(* IEC 61131-3 sources: Word/plc-course/02-electrical-and-field-devices/labs/solutions, 3 files *)

(* ---- 02-1-fail-safe-motor.st ---- *)
(* Lab 02-1: Fail-safe motor circuit - NC stop and overload contacts.
   Module 02 (Electrical fundamentals and field devices).
   REFERENCE SOLUTION - try the lab yourself first.
   Training exercise only: a real machine's emergency stop and safety
   functions are hard-wired or use safety-rated devices (Module 20). *)

PROGRAM FailSafeMotor
  VAR (* I/O - addresses follow the OpenPLC convention *)
    StartPB       AT %IX0.0 : BOOL;  (* Start push-button -S2, NO: TRUE while pressed *)
    StopPB_NC     AT %IX0.1 : BOOL;  (* Stop push-button -S1, NC: TRUE while NOT pressed *)
    OverloadOK_NC AT %IX0.2 : BOOL;  (* Overload relay -F2 contact 95-96, NC: TRUE while healthy *)
    Motor         AT %QX0.0 : BOOL;  (* Motor contactor -Q1 coil (through an interposing relay) *)
    TripLamp      AT %QX0.1 : BOOL;  (* Amber "overload tripped" lamp -H2 *)
  END_VAR

  (* Both NC inputs read TRUE when everything is healthy. A pressed button, a
     tripped overload, a broken wire, a loose terminal or a blown fuse all make
     them read FALSE, so every one of those faults stops the motor. That is
     the point of NC wiring: the "healthy" state has to be actively proven by
     current flowing, so any break in the circuit fails safe.

     Seal-in with both stop conditions in series (AND) with the whole rung:
     when either NC input goes FALSE, Motor drops out and the seal-in is lost.
     When the overload is reset later, nothing restarts: Motor is FALSE and
     only a fresh press of Start can set it again. *)
  Motor := (StartPB OR Motor) AND StopPB_NC AND OverloadOK_NC;

  (* The lamp shows the overload (or its wiring) is not healthy. *)
  TripLamp := NOT OverloadOK_NC;
END_PROGRAM

CONFIGURATION Config0
  RESOURCE Res0 ON PLC
    TASK MainTask(INTERVAL := T#10ms, PRIORITY := 0);
    PROGRAM Inst0 WITH MainTask : FailSafeMotor;
  END_RESOURCE
END_CONFIGURATION

(* ---- 02-2-solenoid-valves.st ---- *)
(* Lab 02-2: Solenoid valves - single-solenoid spring-return versus
   double-solenoid (bistable) valves on the same transfer line.
   Module 02 (Electrical fundamentals and field devices).
   REFERENCE SOLUTION - try the lab yourself first.
   Training exercise only: a real high-high level trip is a safety function
   and would be engineered separately (Module 20). *)

PROGRAM SolenoidValves
  VAR (* I/O - addresses follow the OpenPLC convention *)
    OpenPB         AT %IX0.0 : BOOL;  (* "Open line" push-button, NO: TRUE while pressed *)
    ClosePB_NC     AT %IX0.1 : BOOL;  (* "Close line" push-button, NC: TRUE while NOT pressed *)
    HighLevelOK_NC AT %IX0.2 : BOOL;  (* LSHH on the receiving tank, NC: TRUE while level is NOT high-high *)
    XV201_Sol      AT %QX0.0 : BOOL;  (* XV-201 solenoid: single-solenoid, spring return, fail closed *)
    XV202_OpenSol  AT %QX0.1 : BOOL;  (* XV-202 "open" coil: double-solenoid valve, stays put (fail last) *)
    XV202_CloseSol AT %QX0.2 : BOOL;  (* XV-202 "close" coil *)
  END_VAR
  VAR (* internal *)
    LineOpenCmd : BOOL;  (* TRUE = the line should be open *)
  END_VAR

  (* One command for the line, with a seal-in. Close and the high-high trip
     are NC inputs in series, so a pressed button, a high-high level or a
     broken wire all drop the command. When the trip clears, the command stays
     FALSE until an operator presses Open again: no automatic re-opening. *)
  LineOpenCmd := (OpenPB OR LineOpenCmd) AND ClosePB_NC AND HighLevelOK_NC;

  (* Single-solenoid, spring-return valve: energised = open. The output must
     stay on for as long as the valve is to be open; removing it (by the
     program, by the PLC stopping, or by a power cut) lets the spring close
     the valve. That is why this valve type is used for trips. *)
  XV201_Sol := LineOpenCmd;

  (* Double-solenoid valve: de-energising a coil does NOT move it. The PLC must
     actively drive the close coil to close it. Maintained signals are used:
     the coil for the commanded position stays energised, which re-asserts the
     position if someone has used the manual override, and the two coils are
     complementary, so they can never both be on. At power-up LineOpenCmd is
     FALSE, so the PLC drives the valve closed: after a power cut the program
     cannot know where the valve was left. *)
  XV202_OpenSol  := LineOpenCmd;
  XV202_CloseSol := NOT LineOpenCmd;
END_PROGRAM

CONFIGURATION Config0
  RESOURCE Res0 ON PLC
    TASK MainTask(INTERVAL := T#10ms, PRIORITY := 0);
    PROGRAM Inst0 WITH MainTask : SolenoidValves;
  END_RESOURCE
END_CONFIGURATION

(* ---- 02-3-namur-line-fault.st ---- *)
(* Lab 02-3: NAMUR sensor with line-fault detection - turn a switching
   signal plus open-circuit and short-circuit status bits into a validated
   signal and a fault.
   Module 02 (Electrical fundamentals and field devices).
   REFERENCE SOLUTION - try the lab yourself first.
   Training exercise only: this LSH is a control function. An independent
   high-high protection layer would be engineered separately (Module 20). *)

PROGRAM NamurLineFault
  VAR (* I/O - addresses follow the OpenPLC convention *)
    FillSel      AT %IX0.0 : BOOL;  (* Fill selector: TRUE = operator wants the tank filled *)
    SensorOn     AT %IX0.1 : BOOL;  (* LSH-301 via isolator: TRUE = NAMUR current in the ON band = fork dry *)
    WireBreak    AT %IX0.2 : BOOL;  (* Isolator status: open circuit detected (TRUE = fault) *)
    ShortCircuit AT %IX0.3 : BOOL;  (* Isolator status: short circuit detected (TRUE = fault) *)
    ResetPB      AT %IX0.4 : BOOL;  (* Fault reset push-button, NO: TRUE while pressed *)
    InletValve   AT %QX0.0 : BOOL;  (* XV-301 inlet valve solenoid, spring return: TRUE = open *)
    FaultLamp    AT %QX0.1 : BOOL;  (* Amber "LSH-301 line fault" lamp, latched *)
  END_VAR
  VAR (* internal - required by the lab interface *)
    LineFault : BOOL;  (* TRUE while an open or short circuit is present *)
    HighLevel : BOOL;  (* validated high level: TRUE when high OR when the signal cannot be trusted *)
  END_VAR

  (* 1. Signal quality. Either line fault means SensorOn cannot be trusted:
        a broken wire gives no current (reads as "wet"), and a short circuit
        gives a high current (reads as "dry", the DANGEROUS direction). *)
  LineFault := WireBreak OR ShortCircuit;

  (* 2. Validated signal. The fork is set up fail-safe: current flows while it
        is dry, so a dead sensor reads "wet" = high level. On a line fault the
        program substitutes the safe value, high level, instead of using
        SensorOn. *)
  HighLevel := (NOT SensorOn) OR LineFault;

  (* 3. Latched fault lamp. The fault sets the lamp (and wins while it is
        present). Reset clears it only after the fault has gone, so a brief
        or intermittent fault is still visible to the operator later. *)
  FaultLamp := LineFault OR (FaultLamp AND NOT ResetPB);

  (* 4. Control: fill only when asked to, when the level is known to be below
        the switch, and when no line fault is waiting to be reset.
        - A real high level is a process condition: when the level falls below
          the fork again, filling resumes by itself (a permissive).
        - A line fault is an equipment problem: filling stays stopped until
          someone has looked at it and pressed Reset. That also stops a loose
          terminal from making the valve chatter.
        FaultLamp is worked out above, before it is used here, so the valve
        responds to a reset in the same scan (Module 01: order the program in
        the direction the data flows). *)
  InletValve := FillSel AND NOT HighLevel AND NOT FaultLamp;
END_PROGRAM

CONFIGURATION Config0
  RESOURCE Res0 ON PLC
    TASK MainTask(INTERVAL := T#10ms, PRIORITY := 0);
    PROGRAM Inst0 WITH MainTask : NamurLineFault;
  END_RESOURCE
END_CONFIGURATION
